// TIA Portal project "4Nastri" (V17)
// Vorlageprojekt für das Buch mit Zielsystem S7-1200

(* hardware
DEVICE "S7-1200-Station_1"  S7-1200 Station
   slot 0: "Baugruppenträger_0"  Rack  V1.0
   slot 1: "PLC_1"  CPU 1211C DC/DC/DC  6ES7 211-1AE40-0XB0  V4.1
*)

// ===== PLC "PLC_1"  CPU 1211C DC/DC/DC =====

VAR_GLOBAL   // PLC tag table "Standard-Variablentabelle"
   "S1" AT %I0.0 : Bool;
   "S2" AT %I0.1 : Bool;
   "S3" AT %I0.2 : Bool;
   "S4" AT %I0.3 : Bool;
   "AVA1" AT %Q0.0 : Bool;
   "AVA2" AT %Q0.1 : Bool;
   "AVA3" AT %Q0.2 : Bool;
   "AVA4" AT %Q0.3 : Bool;
END_VAR

DATA_BLOCK "Nastro_Trasportatore_DB"   // DB1
{ S7_Optimized_Access := 'TRUE' }
VERSION : 0.1
// stored: InstanceOfName Nastro_Trasportatore
"Nastro_Trasportatore"
BEGIN
END_DATA_BLOCK

FUNCTION_BLOCK "Nastro"   // FB1, LAD
{ S7_Optimized_Access := 'TRUE' }
VERSION : 0.1
   VAR_INPUT
      S : Bool;
      P_DOPO : Bool;
   END_VAR
   VAR_OUTPUT
      AVA : Bool;
      P_CONS : Bool;
      P_ACC : Bool;
   END_VAR
   VAR
      F0 : Bool;
      F1 : Bool;
      TR0 : Bool;
      TR1 : Bool;
      INIT : Bool;
   END_VAR
BEGIN

REGION Network 1: INIZIALIZZAZIONE
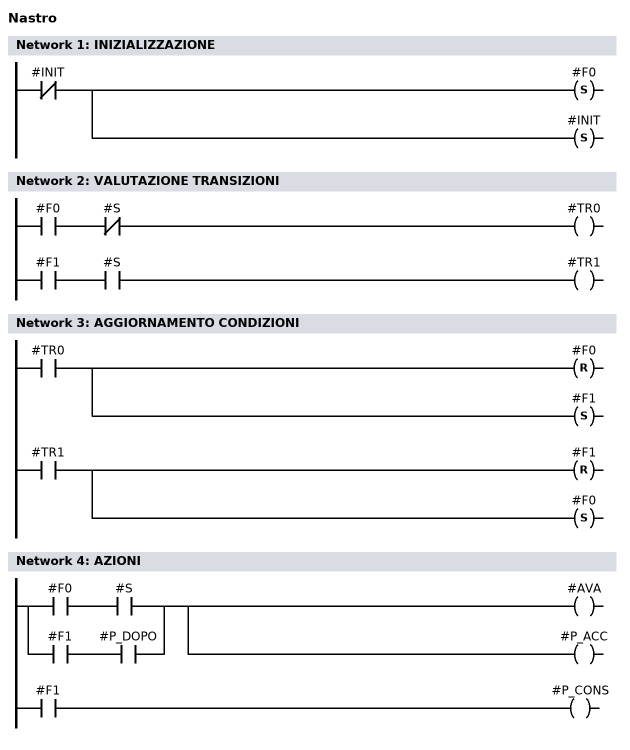
   RUNG wire#powerrail
      I_Contact( #INIT )
      wire#w1
      S_Coil( #F0 )
   END_RUNG
   RUNG wire#w1
      S_Coil( #INIT )
   END_RUNG
   // the same network as SCL:
   IF NOT #INIT THEN
       #F0 := TRUE;
       #INIT := TRUE;
   END_IF;
END_REGION

REGION Network 2: VALUTAZIONE TRANSIZIONI
   RUNG wire#powerrail
      Contact( #F0 )
      I_Contact( #S )
      Coil( #TR0 )
   END_RUNG
   RUNG wire#powerrail
      Contact( #F1 )
      Contact( #S )
      Coil( #TR1 )
   END_RUNG
   // the same network as SCL:
   #TR0 := #F0 AND NOT #S;
   #TR1 := #F1 AND #S;
END_REGION

REGION Network 3: AGGIORNAMENTO CONDIZIONI
   RUNG wire#powerrail
      Contact( #TR0 )
      wire#w1
      R_Coil( #F0 )
   END_RUNG
   RUNG wire#w1
      S_Coil( #F1 )
   END_RUNG
   RUNG wire#powerrail
      Contact( #TR1 )
      wire#w2
      R_Coil( #F1 )
   END_RUNG
   RUNG wire#w2
      S_Coil( #F0 )
   END_RUNG
   // the same network as SCL:
   IF #TR0 THEN
       #F0 := FALSE;
       #F1 := TRUE;
   END_IF;
   IF #TR1 THEN
       #F1 := FALSE;
       #F0 := TRUE;
   END_IF;
END_REGION

REGION Network 4: AZIONI
   RUNG wire#powerrail
      Contact( #F0 )
      Contact( #S )
      wire#w1
      Coil( #AVA )
   END_RUNG
   RUNG wire#powerrail
      Contact( #F1 )
      Contact( #P_DOPO )
   END_RUNG wire#w1
   RUNG wire#w1
      Coil( #P_ACC )
   END_RUNG
   RUNG wire#powerrail
      Contact( #F1 )
      Coil( #P_CONS )
   END_RUNG
   // the same network as SCL:
   #AVA := (#F0 AND #S) OR (#F1 AND #P_DOPO);
   #P_ACC := #AVA;
   #P_CONS := #F1;
END_REGION
END_FUNCTION_BLOCK

FUNCTION_BLOCK "Nastro_Trasportatore"   // FB2, FBD
{ S7_Optimized_Access := 'TRUE' }
VERSION : 0.1
   VAR
      Nastro_Instance : "Nastro";
      Nastro_Instance_1 : "Nastro";
      Nastro_Instance_2 : "Nastro";
      Nastro_Instance_3 : "Nastro";
   END_VAR
   VAR CONSTANT
      TRUE : Bool := true;
      FALSE : Bool;
   END_VAR
BEGIN

REGION Network 1
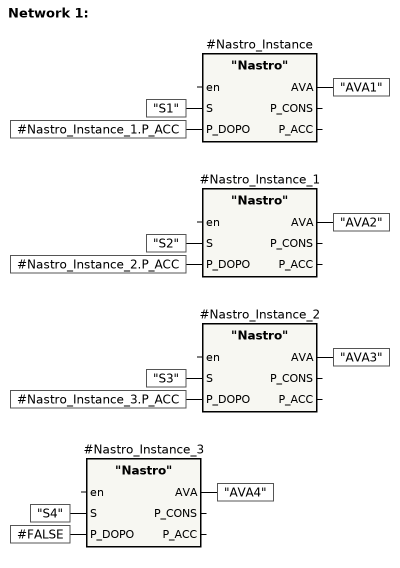
   #Nastro_Instance(S := "S1", P_DOPO := #Nastro_Instance_1.P_ACC, AVA => "AVA1");   // "Nastro"
   #Nastro_Instance_1(S := "S2", P_DOPO := #Nastro_Instance_2.P_ACC, AVA => "AVA2");   // "Nastro"
   #Nastro_Instance_2(S := "S3", P_DOPO := #Nastro_Instance_3.P_ACC, AVA => "AVA3");   // "Nastro"
   #Nastro_Instance_3(S := "S4", P_DOPO := #FALSE, AVA => "AVA4");   // "Nastro"
END_REGION
END_FUNCTION_BLOCK

FUNCTION "MHJ-PLC-Lab-Function-S71200" : Void   // FC9000, SCL
{ S7_Optimized_Access := 'TRUE' }
VERSION : 0.1
   VAR_TEMP
      rdTimeReturn : Int;
      outputTime : DTL;
      SyncVal : Byte;
      forVal : Int;
      forVal_2 : Int;
      Value : Byte;
   END_VAR
   VAR CONSTANT
      CompVal : Byte := 16#34;
      Value_01 : Byte := 16#11;
      Value_01_DW : DWord := 16#A165_D992;
      Value_02_DW : DWord := 16#58BE_4401;
   END_VAR
BEGIN

   #Value:=PEEK(area := 16#82,
        dbNumber := 0,
        byteOffset := 511);
   #Value := #Value + 1;

   POKE(area := 16#82,
        dbNumber := 0,
        byteOffset := 511,
        value := #Value);

   POKE(area:=16#81,
        dbNumber:=0,
        byteOffset:=1016,
        value:=#Value_01_DW);
   POKE(area := 16#81,
        dbNumber := 0,
        byteOffset := 1020,
        value := #Value_02_DW);

   POKE(area := 16#81,
        dbNumber := 0,
        byteOffset := 511,
        value := B#16#00);

   FOR #forVal := 0 TO 120 DO
       FOR #forVal_2:=0 TO 10 DO
           #rdTimeReturn:=RD_SYS_T(#outputTime);
           #rdTimeReturn := WR_SYS_T(#outputTime);
           #rdTimeReturn := RD_SYS_T(#outputTime);
           #rdTimeReturn := WR_SYS_T(#outputTime);
       END_FOR;
       #SyncVal:= PEEK(area := 16#81,
                      dbNumber := 0,
                      byteOffset := 511);
       IF #SyncVal = #CompVal THEN
          GOTO M_1;
       END_IF;
   END_FOR;
   RETURN;

   M_1:
   POKE(area := 16#81,
        dbNumber := 0,
        byteOffset := 511,
        value := B#16#0);
END_FUNCTION

ORGANIZATION_BLOCK "Main"   // OB1, FBD, ProgramCycle
TITLE = "Main Program Sweep (Cycle)"
{ S7_Optimized_Access := 'TRUE' }
VERSION : 0.1
   VAR_INPUT
      Initial_Call : Bool;   // Initial call of this OB
      Remanence : Bool;   // =True, if remanent data are available
   END_VAR
BEGIN

REGION Network 1: Konnektierungsbaustein für PLC-Lab
   // Im Netzwerk 1 wird der Konnektierungsbaustein für PLC-Lab aufgerufen.
   // Dieser Aufruf darf nicht entfernt werden!
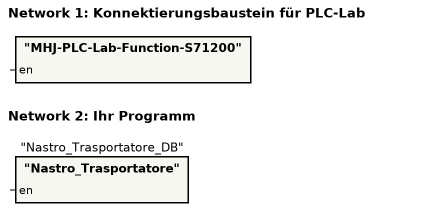
   "MHJ-PLC-Lab-Function-S71200"();
END_REGION

REGION Network 2: Ihr Programm
   // Schreiben Sie ab Netzwerk 2 Ihr Programm
   "Nastro_Trasportatore_DB"();   // "Nastro_Trasportatore"
END_REGION
END_ORGANIZATION_BLOCK